// SIMATIC S7-200 project (STEP 7-Micro/WIN), CPU 221 REL 01.10

ORGANIZATION_BLOCK PRINCIPAL:OB1
TITLE=MONOESTABLE CON RESET  /  JEVG
BEGIN
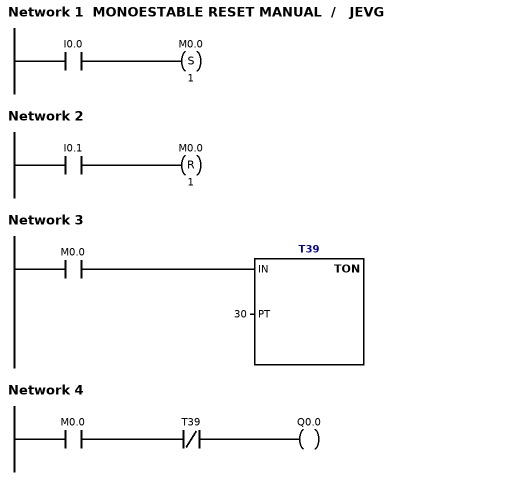
Network 1 // MONOESTABLE RESET MANUAL  /   JEVG
LD     I0.0
S      M0.0, 1
Network 2
LD     I0.1
R      M0.0, 1
Network 3
LD     M0.0
TON    T39, 30
Network 4
LD     M0.0
AN     T39
=      Q0.0
END_ORGANIZATION_BLOCK
